Yaskawa INFORM job: clamp_cylinder_program.JBI

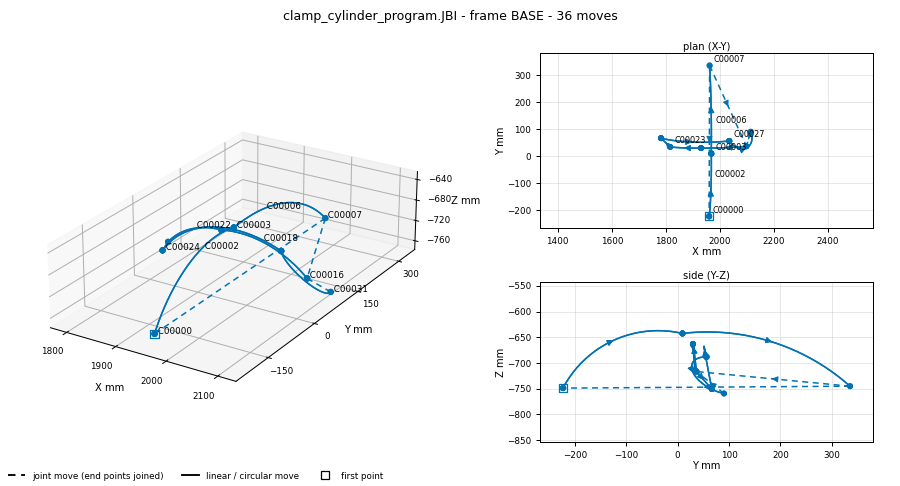
[picture p0: tool path of clamp_cylinder_program.JBI in frame BASE, 36 of 54 moves have a stored position in this frame; points joined in program order, loops and branches not executed]
/JOB
//NAME clamp_cylinder_program
//POS
///NPOS 48,0,48,0,0,0
///TOOL 0
///POSTYPE BASE
///RECTAN
///RCONF 0,0,0,0,0,0,0,0,0,0,0,0,0,0,0,0,0,0,0,0,0,0,0,0
C00000=1960.301339,-223.020258,-748.833463,180.000000,-60.000000,90.001386
C00001=1960.301339,-223.020258,-748.833463,180.000000,-60.000000,90.001386
C00002=1967.903284,-90.586140,-643.796844,-152.219285,5.000000,5.000000
C00003=1968.241109,9.331558,-642.480132,-175.000000,5.000000,5.000000
C00004=1968.241109,9.331558,-642.480132,-175.000000,5.000000,5.000000
C00005=1968.241109,9.331558,-642.480132,-175.000000,5.000000,5.000000
C00006=1968.519242,106.958551,-642.493976,154.871761,5.000000,-5.000000
C00007=1961.960608,335.261942,-745.099188,-180.000000,-60.000000,-90.296572
C00008=1960.301339,-223.020258,-748.833463,180.000000,-60.000000,90.001386
C00009=1960.301339,-223.020258,-748.833463,180.000000,-60.000000,90.001386
C00010=1967.903284,-90.586140,-643.796844,-152.219285,5.000000,5.000000
C00011=1968.241109,9.331558,-642.480132,-175.000000,5.000000,5.000000
C00012=1968.241109,9.331558,-642.480132,-175.000000,5.000000,5.000000
C00013=1968.241109,9.331558,-642.480132,-175.000000,5.000000,5.000000
C00014=1968.519242,106.958551,-642.493976,154.871761,5.000000,-5.000000
C00015=1961.960608,335.261942,-745.099188,-180.000000,-60.000000,-90.296572
C00016=2098.047200,36.518447,-716.632227,-175.000000,-47.125831,175.000000
C00017=2098.047200,36.518447,-716.632227,-175.000000,-47.125831,175.000000
C00018=2009.615266,30.727639,-665.973209,-174.277481,14.920308,5.000000
C00019=1930.361446,29.759393,-663.154630,-174.166812,-9.802458,-5.000000
C00020=1930.361446,29.759393,-663.154630,-174.166812,-9.802458,-5.000000
C00021=1930.361446,29.759393,-663.154630,-174.166812,-9.802458,-5.000000
C00022=1873.200556,30.292187,-673.540133,-173.338787,-27.257617,-5.000000
C00023=1816.362021,33.789116,-713.796526,175.000000,-48.409654,5.545682
C00024=1782.142124,66.487085,-750.681160,-180.000000,-60.000000,1.268197
C00025=1782.142124,66.487085,-750.681160,-180.000000,-60.000000,1.268197
C00026=1861.781127,54.155854,-685.576790,175.000000,-33.017894,9.272615
C00027=2034.789788,55.906022,-688.063230,-173.996373,25.294573,5.000000
C00028=2034.789788,55.906022,-688.063230,-173.996373,25.294573,5.000000
C00029=2034.789788,55.906022,-688.063230,-173.996373,25.294573,5.000000
C00030=2118.765899,62.702710,-749.259165,175.000000,-59.670456,175.000000
C00031=2114.208826,90.160050,-759.297271,-180.000000,-60.000000,-172.642433
C00032=2098.047200,36.518447,-716.632227,-175.000000,-47.125831,175.000000
C00033=2098.047200,36.518447,-716.632227,-175.000000,-47.125831,175.000000
C00034=2009.615266,30.727639,-665.973209,-174.277481,14.920308,5.000000
C00035=1930.361446,29.759393,-663.154630,-174.166812,-9.802458,-5.000000
C00036=1930.361446,29.759393,-663.154630,-174.166812,-9.802458,-5.000000
C00037=1930.361446,29.759393,-663.154630,-174.166812,-9.802458,-5.000000
C00038=1873.200556,30.292187,-673.540133,-173.338787,-27.257617,-5.000000
C00039=1816.362021,33.789116,-713.796526,175.000000,-48.409654,5.545682
C00040=1782.142124,66.487085,-750.681160,-180.000000,-60.000000,1.268197
C00041=1782.142124,66.487085,-750.681160,-180.000000,-60.000000,1.268197
C00042=1861.781127,54.155854,-685.576790,175.000000,-33.017894,9.272615
C00043=2034.789788,55.906022,-688.063230,-173.996373,25.294573,5.000000
C00044=2034.789788,55.906022,-688.063230,-173.996373,25.294573,5.000000
C00045=2034.789788,55.906022,-688.063230,-173.996373,25.294573,5.000000
C00046=2118.765899,62.702710,-749.259165,175.000000,-59.670456,175.000000
C00047=2114.208826,90.160050,-759.297271,-180.000000,-60.000000,-172.642433
///POSTYPE PULSE
///PULSE
EX00000=0
EX00001=92160
EX00002=184320
EX00003=276480
///POSTYPE PULSE
///PULSE
EC00000=0
EC00001=0
EC00002=0
EC00003=0
EC00004=0
EC00005=0
EC00006=0
EC00007=0
EC00008=0
EC00009=0
EC00010=0
EC00011=0
EC00012=0
EC00013=0
EC00014=0
EC00015=0
EC00016=0
EC00017=0
EC00018=0
EC00019=0
EC00020=0
EC00021=0
EC00022=0
EC00023=0
EC00024=0
EC00025=0
EC00026=0
EC00027=0
EC00028=0
EC00029=0
EC00030=0
EC00031=0
EC00032=0
EC00033=0
EC00034=0
EC00035=0
EC00036=0
EC00037=0
EC00038=0
EC00039=0
EC00040=0
EC00041=0
EC00042=0
EC00043=0
EC00044=0
EC00045=0
EC00046=0
EC00047=0
//INST
///DATE 2023/08/07 12:27
///ATTR SC,RW,RJ
////FRAME BASE
///GROUP1 RB1,ST1
NOP
MOVJ P009 EX000 VJ=15.00
MOVJ C00000 EC00000 VJ=15.0
CALL JOB:SPYON
MOVC C00001 EC00001 V=150.0
MOVC C00002 EC00002 V=150.0
MOVC C00003 EC00003 V=150.0
MOVL C00004 EC00004 V=150.0
MOVC C00005 EC00005 V=150.0
MOVC C00006 EC00006 V=150.0
MOVC C00007 EC00007 V=150.0
CALL JOB:SPYOF
MOVJ C00008 EC00008 VJ=15.0
CALL JOB:SPYON
MOVC C00009 EC00009 V=150.0
MOVC C00010 EC00010 V=150.0
MOVC C00011 EC00011 V=150.0
MOVL C00012 EC00012 V=150.0
MOVC C00013 EC00013 V=150.0
MOVC C00014 EC00014 V=150.0
MOVC C00015 EC00015 V=150.0
CALL JOB:SPYOF
MOVJ C00016 EC00016 VJ=15.0
CALL JOB:SPYON
MOVC C00017 EC00017 V=150.0
MOVC C00018 EC00018 V=150.0
MOVC C00019 EC00019 V=150.0
MOVL C00020 EC00020 V=150.0
MOVC C00021 EC00021 V=150.0
MOVC C00022 EC00022 V=150.0
MOVC C00023 EC00023 V=150.0
MOVL C00024 EC00024 V=150.0
MOVC C00025 EC00025 V=150.0
MOVC C00026 EC00026 V=150.0
MOVC C00027 EC00027 V=150.0
MOVL C00028 EC00028 V=150.0
MOVC C00029 EC00029 V=150.0
MOVC C00030 EC00030 V=150.0
MOVC C00031 EC00031 V=150.0
CALL JOB:SPYOF
MOVJ C00032 EC00032 VJ=15.0
CALL JOB:SPYON
MOVC C00033 EC00033 V=150.0
MOVC C00034 EC00034 V=150.0
MOVC C00035 EC00035 V=150.0
MOVL C00036 EC00036 V=150.0
MOVC C00037 EC00037 V=150.0
MOVC C00038 EC00038 V=150.0
MOVC C00039 EC00039 V=150.0
MOVL C00040 EC00040 V=150.0
MOVC C00041 EC00041 V=150.0
MOVC C00042 EC00042 V=150.0
MOVC C00043 EC00043 V=150.0
MOVL C00044 EC00044 V=150.0
MOVC C00045 EC00045 V=150.0
MOVC C00046 EC00046 V=150.0
MOVC C00047 EC00047 V=150.0
CALL JOB:SPYOF
MOVJ P009 VJ=15.00
MOVJ P009 VJ=15.00
MOVJ P009 VJ=15.00
MOVJ P009 VJ=15.00
MOVJ P009 VJ=15.00
END
